// TIA Portal V20 export
TYPE "LER_typeBrakeTestEmMonitoring"
// stored: Access Published
   STRUCT
      error { ExternalWritable := 'False'} : Bool;
      ready { ExternalWritable := 'False'} : Bool;
      busy { ExternalWritable := 'False'} : Bool;
      complete { ExternalWritable := 'False'} : Bool;
      brakeSelected { ExternalWritable := 'False'} : Bool;
      brakeActive { ExternalWritable := 'False'} : Bool;
      brakeResult { ExternalWritable := 'False'} : Bool;
      brakeCompleted { ExternalWritable := 'False'} : Bool;
      "step" { ExternalWritable := 'False'} : Int;
   END_STRUCT;
END_TYPE
